// TIA Portal V16 program export: 0 tag tables, 1 data types, 0 data blocks, 3 code blocks (in call order from the OBs), 0 instance data blocks

TYPE "Message_UDT"
// stored: IsFailsafeCompliant false
   STRUCT
      String_1 : WString;
      String_2 : WString;
      String_3 : WString;
      String_4 : WString;
   END_STRUCT;
END_TYPE

ORGANIZATION_BLOCK "Main"   // OB1, LAD, ProgramCycle
TITLE = "Main Program Sweep (Cycle)"
{ S7_Optimized_Access := 'TRUE' }
VERSION : 0.1
// stored: AutoNumber true, IsIECCheckEnabled false, SetENOAutomatically false
   VAR_INPUT
      Initial_Call : Bool;   // Initial call of this OB
      Remanence : Bool;   // =True, if remanent data are available
   END_VAR
BEGIN

NETWORK
TITLE = 



      A     "Tag_1";
      =     "Tag_2";




END_ORGANIZATION_BLOCK

FUNCTION "Test_AWL" : Void   // FC2, STL
{ S7_Optimized_Access := 'TRUE' }
VERSION : 0.1
// stored: AutoNumber true, UDAEnableTagReadback false
   VAR_TEMP
      x_Test_1 : Bool;
      x_Test_2 : Bool;
      x_Test_3 : Bool;
      x_Test_4 : Bool;
      x_Test_5 : Bool;
   END_VAR
BEGIN

NETWORK
TITLE = 
      A     #x_Test_1;
      =     #x_Test_2;

END_FUNCTION

FUNCTION "Message" : Void
{ S7_Optimized_Access := 'TRUE' }
VERSION : 0.1
   VAR_INPUT 
      IN_WString : WString;
   END_VAR

   VAR_OUTPUT 
      OUT_WString : WString;
   END_VAR

   VAR_IN_OUT 
      Cache : "Message_UDT";
   END_VAR


BEGIN
	REGION _name_
	    #OUT_WString := #IN_WString;
	END_REGION
	
	
	
	
	
	
	
END_FUNCTION
